{attribute 'GeneratedUsingTerminal: ER3204-0002-0016'}
{attribute addProperty BoxType "ER3204-0002-0016"}
{attribute addProperty Id "RTD_RTDInputs_Channel_1AT %I*RTD_RTDInputs_Channel_A8DF64E310RTD_RTDInputs_Channel_2AT %I*RTD_RTDInputs_Channel_A8DF64E310RTD_RTDInputs_Channel_3AT %I*RTD_RTDInputs_Channel_A8DF64E310RTD_RTDInputs_Channel_4AT %I*RTD_RTDInputs_Channel_A8DF64E310WcStateAT %I*WcState_9091E0EB2InfoDataAT %I*InfoData_94A18F5E2"}
{attribute addProperty CRC "161035556"}
{attribute addProperty Size "44"}
TYPE ER3204_09993524 EXTENDS EtcSlaveTerminalBase_947E5A46 :
STRUCT
	{attribute addProperty Name "RTD_RTDInputs_Channel_1"}
	RTD_RTDInputs_Channel_1 : RTD_RTDInputs_Channel_A8DF64E3;
	{attribute addProperty Name "RTD_RTDInputs_Channel_2"}
	RTD_RTDInputs_Channel_2 : RTD_RTDInputs_Channel_A8DF64E3;
	{attribute addProperty Name "RTD_RTDInputs_Channel_3"}
	RTD_RTDInputs_Channel_3 : RTD_RTDInputs_Channel_A8DF64E3;
	{attribute addProperty Name "RTD_RTDInputs_Channel_4"}
	RTD_RTDInputs_Channel_4 : RTD_RTDInputs_Channel_A8DF64E3;
	{attribute addProperty Name "WcState"}
	WcState : WcState_9091E0EB;
	{attribute addProperty Name "InfoData"}
	InfoData : InfoData_94A18F5E;
END_STRUCT
END_TYPE

(* stored: Version 1.2.0.0, ProductVersion 3.1.4024.9
   DUT ER3204_09993524: Id {4fb9abe7-d12e-4411-af1a-51f99dbe81bc} *)
